PROGRAM MAIN
VAR
END_VAR

END_PROGRAM

(* stored: Version 1.1.0.1
   POU MAIN: Id {f8d99e63-1973-4a2f-827e-afffdbd00bdc} *)
